// TIA Portal V20 export
DATA_BLOCK "2000_Motion"   // DB450
// stored: MemoryReserve 100
   VAR
      Dancer : Struct
         Commands : Struct
            Enable : Bool;
            Stop : Bool;
            Reset : Bool;
         END_STRUCT;
         Parameters : Struct
            DancerDirection : Bool;
            UnWinderDirection : Bool;
            UnwinderTopUse : Bool;
            UnwinderBottomUse : Bool;
            JogMode : Bool;
            SetPoint : LReal;
            Input : LReal;
            Kp : LReal;
            Ki : LReal;
            Radius : LReal;
         END_STRUCT;
         Status : Struct
            StopRequest : Bool;
            Busy : Struct
               TotalBusy : Bool;
               EnableBusy : Bool;
               StopBusy : Bool;
               ResetBusy : Bool;
            END_STRUCT;
            Done : Struct
               TotalDone : Bool;
               EnableDone : Bool;
               StopDone : Bool;
               ResetDone : Bool;
            END_STRUCT;
            Error : Bool;
            ErrorID : DWord;
            StatusID : DWord;
            NowCmd : DInt;
            BeforeCmd : DInt;
            NowStep : DInt;
            BeforeStep : DInt;
         END_STRUCT;
      END_STRUCT;
      StackMain : Struct
         Commands : Struct
            Calculate : Bool := FALSE;
            SemiStep : Bool := FALSE;
            FullStep : Bool := FALSE;
            Auto : Bool := FALSE;
            CycleStop : Bool := FALSE;
            FastStop : Bool := FALSE;
            Reset : Bool := FALSE;
         END_STRUCT;
         Parameters : Struct
            Global : Struct
               CPM : LReal := 10.0;
               StageWidth : LReal := 244.14;
            END_STRUCT;
            "Step" : Struct
               MandrelUse : Bool;
               InitialPosFinalRoller : LReal := 0.0;
               InitialPosCompensator : LReal := 0.0;
            END_STRUCT;
            Auto : Struct
               SepaClean : Bool;
               CellCount : DInt;
               Compensator : Struct
                  InitialPosCompensator : LReal;
               END_STRUCT;
               Anode : Struct
                  PnPX1 : Struct
                     InitialPosAnodePnPX1 : LReal;
                     AnodePnPX1FwdOutputCam : Struct
                        OnPos : LReal := 10.0;
                        OffPos : LReal := 530.0;
                     END_STRUCT;
                     AnodePnPX1BwdOutputCam : Struct
                        OnPos : LReal := 10.0;
                        OffPos : LReal := 530.0;
                     END_STRUCT;
                     AnodeReelCutDataDeleteOffOutputCam : Struct
                        OnPos : LReal := 10.0;
                        OffPos : LReal := 530.0;
                     END_STRUCT;
                  END_STRUCT;
                  PnPX2 : Struct
                     InitialPosAnodePnPX2 : LReal;
                     AnodePnPX2FwdOutputCam : Struct
                        OnPos : LReal := 10.0;
                        OffPos : LReal := 530.0;
                     END_STRUCT;
                     AnodePnPX2BwdOutputCam : Struct
                        OnPos : LReal := 10.0;
                        OffPos : LReal := 530.0;
                     END_STRUCT;
                  END_STRUCT;
                  PnPZ1 : Struct
                     InitialPosAnodePnPZ1 : LReal := 0.0;
                     AnodePnPZ1Down1OutputCam : Struct
                        OnPos : LReal := 1.0;
                        OffPos : LReal := 24.0;
                     END_STRUCT;
                     AnodePnPZ1Up1OutputCam : Struct
                        OnPos : LReal := 1.0;
                        OffPos : LReal := 24.0;
                     END_STRUCT;
                     AnodePnPZ1Down2OutputCam : Struct
                        OnPos : LReal := 1.0;
                        OffPos : LReal := 29.0;
                     END_STRUCT;
                     AnodePnPZ1Up2OutputCam : Struct
                        OnPos : LReal := 1.0;
                        OffPos : LReal := 29.0;
                     END_STRUCT;
                     AnodePnPZ1SuctionOnOutputCam : Struct
                        OnPos : LReal := 23.0;
                        OffPos : LReal := 28.0;
                     END_STRUCT;
                     AnodePnPZ1SuctionOffOutputCam : Struct
                        OnPos : LReal := 23.0;
                        OffPos : LReal := 30.0;
                     END_STRUCT;
                     AnodePnPZ1ReelCutBlowOutputCam : Struct
                        OnPos : LReal := 22.0;
                        OffPos : LReal := 28.0;
                     END_STRUCT;
                     AnodeAlignSuctionOnOutputCam : Struct
                        OnPos : LReal := 22.0;
                        OffPos : LReal := 30.0;
                     END_STRUCT;
                     AnodeReelCutDataDeleteOnOutputCam : Struct
                        OnPos : LReal := 5.0;
                        OffPos : LReal := 20.0;
                     END_STRUCT;
                     AnodeAlignVisionOutputCam : Struct
                        OnPos : LReal := 1.0;
                        OffPos : LReal := 24.0;
                     END_STRUCT;
                  END_STRUCT;
                  PnPZ2 : Struct
                     InitialPosAnodePnPZ2 : LReal := 0.0;
                     AnodePnPZ2Down1OutputCam : Struct
                        OnPos : LReal := 1.0;
                        OffPos : LReal := 24.0;
                     END_STRUCT;
                     AnodePnPZ2Up1OutputCam : Struct
                        OnPos : LReal := 1.0;
                        OffPos : LReal := 24.0;
                     END_STRUCT;
                     AnodePnPZ2Down2OutputCam : Struct
                        OnPos : LReal := 1.0;
                        OffPos : LReal := 29.0;
                     END_STRUCT;
                     AnodePnPZ2Up2OutputCam : Struct
                        OnPos : LReal := 1.0;
                        OffPos : LReal := 29.0;
                     END_STRUCT;
                     AnodePnPZ2SuctionOnOutputCam : Struct
                        OnPos : LReal := 23.0;
                        OffPos : LReal := 30.0;
                     END_STRUCT;
                     AnodePnPZ2SuctionOffOutputCam : Struct
                        OnPos : LReal := 22.0;
                        OffPos : LReal := 28.0;
                     END_STRUCT;
                     AnodeAlignSuctionOffOutputCam : Struct
                        OnPos : LReal := 22.0;
                        OffPos : LReal := 30.0;
                     END_STRUCT;
                  END_STRUCT;
               END_STRUCT;
               Cathode : Struct
                  PnPX1 : Struct
                     InitialPosCathodePnPX1 : LReal;
                     CathodePnPX1FwdOutputCam : Struct
                        OnPos : LReal := 10.0;
                        OffPos : LReal := 530.0;
                     END_STRUCT;
                     CathodePnPX1BwdOutputCam : Struct
                        OnPos : LReal := 10.0;
                        OffPos : LReal := 530.0;
                     END_STRUCT;
                     CathodeReelCutDataDeleteOffOutputCam : Struct
                        OnPos : LReal := 10.0;
                        OffPos : LReal := 530.0;
                     END_STRUCT;
                  END_STRUCT;
                  PnPX2 : Struct
                     InitialPosCathodePnPX2 : LReal;
                     CathodePnPX2FwdOutputCam : Struct
                        OnPos : LReal := 10.0;
                        OffPos : LReal := 530.0;
                     END_STRUCT;
                     CathodePnPX2BwdOutputCam : Struct
                        OnPos : LReal := 10.0;
                        OffPos : LReal := 530.0;
                     END_STRUCT;
                  END_STRUCT;
                  PnPZ1 : Struct
                     InitialPosCathodePnPZ1 : LReal;
                     CathodePnPZ1Down1OutputCam : Struct
                        OnPos : LReal := 1.0;
                        OffPos : LReal := 24.0;
                     END_STRUCT;
                     CathodePnPZ1Up1OutputCam : Struct
                        OnPos : LReal := 1.0;
                        OffPos : LReal := 24.0;
                     END_STRUCT;
                     CathodePnPZ1Down2OutputCam : Struct
                        OnPos : LReal := 1.0;
                        OffPos : LReal := 29.0;
                     END_STRUCT;
                     CathodePnPZ1Up2OutputCam : Struct
                        OnPos : LReal := 1.0;
                        OffPos : LReal := 29.0;
                     END_STRUCT;
                     CathodePnPZ1SuctionOnOutputCam : Struct
                        OnPos : LReal := 23.0;
                        OffPos : LReal := 28.0;
                     END_STRUCT;
                     CathodePnPZ1SuctionOffOutputCam : Struct
                        OnPos : LReal := 23.0;
                        OffPos : LReal := 30.0;
                     END_STRUCT;
                     CathodePnPZ1ReelCutBlowOutputCam : Struct
                        OnPos : LReal := 22.0;
                        OffPos : LReal := 28.0;
                     END_STRUCT;
                     CathodeAlignSuctionOnOutputCam : Struct
                        OnPos : LReal := 22.0;
                        OffPos : LReal := 30.0;
                     END_STRUCT;
                     CathodeReelCutDataDeleteOnOutputCam : Struct
                        OnPos : LReal := 5.0;
                        OffPos : LReal := 20.0;
                     END_STRUCT;
                     CathodeAlignVisionOutputCam : Struct
                        OnPos : LReal := 1.0;
                        OffPos : LReal := 24.0;
                     END_STRUCT;
                  END_STRUCT;
                  PnPZ2 : Struct
                     InitialPosCathodePnPZ2 : LReal;
                     CathodePnPZ2Down1OutputCam : Struct
                        OnPos : LReal := 1.0;
                        OffPos : LReal := 24.0;
                     END_STRUCT;
                     CathodePnPZ2Up1OutputCam : Struct
                        OnPos : LReal := 1.0;
                        OffPos : LReal := 24.0;
                     END_STRUCT;
                     CathodePnPZ2Down2OutputCam : Struct
                        OnPos : LReal := 1.0;
                        OffPos : LReal := 29.0;
                     END_STRUCT;
                     CathodePnPZ2Up2OutputCam : Struct
                        OnPos : LReal := 1.0;
                        OffPos : LReal := 29.0;
                     END_STRUCT;
                     CathodePnPZ2SuctionOnOutputCam : Struct
                        OnPos : LReal := 23.0;
                        OffPos : LReal := 28.0;
                     END_STRUCT;
                     CathodePnPZ2SuctionOffOutputCam : Struct
                        OnPos : LReal := 23.0;
                        OffPos : LReal := 30.0;
                     END_STRUCT;
                     CathodeAlignSuctionOffOutputCam : Struct
                        OnPos : LReal := 22.0;
                        OffPos : LReal := 30.0;
                     END_STRUCT;
                  END_STRUCT;
               END_STRUCT;
               FinalRoller : Struct
                  InitialPosFinalRoller : LReal;
                  FinalRollerFwdOutputCam : Struct
                     OnPos : LReal := 10.0;
                     OffPos : LReal := 330.0;
                  END_STRUCT;
                  FinalRollerBwdOutputCam : Struct
                     OnPos : LReal := 10.0;
                     OffPos : LReal := 330.0;
                  END_STRUCT;
                  FinalRollerStackTableDownOutputCam : Struct
                     OnPos : LReal := 140.0;
                     OffPos : LReal := 200.0;
                  END_STRUCT;
                  FinalRollerStackAnodeVisionOutputCam : Struct
                     OnPos : LReal := 10.0;
                     OffPos : LReal := 40.0;
                  END_STRUCT;
                  FinalRollerStackCathodeVisionOutputCam : Struct
                     OnPos : LReal := 300.0;
                     OffPos : LReal := 330.0;
                  END_STRUCT;
               END_STRUCT;
               Mandrel : Struct
                  InitialPosAnodeMandrelYFront : LReal;
                  InitialPosAnodeMandrelYRear : LReal;
                  InitialPosAnodeMandrelZFront : LReal;
                  InitialPosAnodeMandrelZRear : LReal;
                  InitialPosCathodeMandrelYFront : LReal;
                  InitialPosCathodeMandrelYRear : LReal;
                  InitialPosCathodeMandrelZFront : LReal;
                  InitialPosCathodeMandrelZRear : LReal;
               END_STRUCT;
            END_STRUCT;
            StackCalculate : Struct
               Direction : Bool := TRUE;
               RatioOption : Bool := TRUE;
               TimeOption : Bool;
               PosOption : Bool;
               DoubleOption : Bool;
               StageHeight : LReal := 360.0;
               StageGap : LReal := 5.0;
               AccRatio : DInt := 3;
               Ratio : Struct
                  FinalRollerStart : LReal := 0.0;
                  FinalRollerEnd : LReal := 75.0;
                  PnPXStart : LReal := 0.0;
                  PnPXEnd : LReal := 75.0;
                  PnPZDownStart : LReal := 65.0;
                  PnPZDownEnd : LReal := 75.0;
                  PnPZUpStart : LReal := 90.0;
                  PnPZUpEnd : LReal := 100.0;
                  MandrelBwdStart : LReal := 75.0;
                  MandrelBwdEnd : LReal := 82.5;
                  MandrelFwdStart : LReal := 82.5;
                  MandrelFwdEnd : LReal := 90.0;
                  MandrelUpStart1 : LReal := 55.0;
                  MandrelUpEnd1 : LReal := 62.5;
                  MandrelUpStart2 : LReal := 75.0;
                  MandrelUpEnd2 : LReal := 82.5;
                  MandrelDownStart : LReal := 87.0;
                  MandrelDownEnd : LReal := 90.0;
                  MandrelYTerm : LReal := 0.0;
                  MandrelZTerm : LReal := 0.0;
                  MandrelBwdOffset : LReal := 0.0;
                  MandrelFwdOffset : LReal := 0.0;
               END_STRUCT;
               "Time" : Struct
                  FinalRollerStart : LReal;
                  FinalRollerEnd : LReal;
                  PnPXStart : LReal;
                  PnPXEnd : LReal;
                  PnPZDownStart : LReal;
                  PnPZDownEnd : LReal;
                  PnPZUpStart : LReal;
                  PnPZUpEnd : LReal;
                  MandrelBwdStart : LReal;
                  MandrelBwdEnd : LReal;
                  MandrelFwdStart : LReal;
                  MandrelFwdEnd : LReal;
                  MandrelUpStart1 : LReal;
                  MandrelUpEnd1 : LReal;
                  MandrelUpStart2 : LReal;
                  MandrelUpEnd2 : LReal;
                  MandrelDownStart : LReal;
                  MandrelDownEnd : LReal;
               END_STRUCT;
               Position : Struct
                  FinalRollerBwdPos : LReal;
                  FinalRollerFwdPos : LReal;
               END_STRUCT;
               Distance : Struct
                  Compensator : Struct
                     Null : Bool;
                  END_STRUCT;
                  Anode : Struct
                     PnPX1Distance : LReal := 540.0;
                     PnPX2Distance : LReal := 540.0;
                     PnPZ1Distance1 : LReal := 25.0;
                     PnPZ1Distance2 : LReal := 27.0;
                     PnPZ2Distance1 : LReal := 25.0;
                     PnPZ2Distance2 : LReal := 27.0;
                  END_STRUCT;
                  Cathode : Struct
                     PnPX1Distance : LReal := 540.0;
                     PnPX2Distance : LReal := 540.0;
                     PnPZ1Distance1 : LReal := 25.0;
                     PnPZ1Distance2 : LReal := 27.0;
                     PnPZ2Distance1 : LReal := 25.0;
                     PnPZ2Distance2 : LReal := 27.0;
                  END_STRUCT;
                  FinalRoller : Struct
                     Distance : LReal := 350.0;
                  END_STRUCT;
                  Mandrel : Struct
                     AnodeMandrelYFrontDistance : LReal := 20.0;
                     AnodeMandrelYRearDistance : LReal := 20.0;
                     CathodeMandrelYFrontDistance : LReal := 20.0;
                     CathodeMandrelYRearDistance : LReal := 20.0;
                     AnodeMandrelZFrontDistance : LReal := 10.0;
                     AnodeMandrelZRearDistance : LReal := 10.0;
                     CathodeMandrelZFrontDistance : LReal := 10.0;
                     CathodeMandrelZRearDistance : LReal := 10.0;
                  END_STRUCT;
               END_STRUCT;
            END_STRUCT;
         END_STRUCT;
         Status : Struct
            StopRequest : Bool;
            Busy : Struct
               TotalBusy : Bool;
               CalculateBusy : Bool;
               SemiStepBusy : Bool;
               FullStepBusy : Bool;
               AutoBusy : Bool;
               CycleStopBusy : Bool;
               FastStopBusy : Bool;
               ResetBusy : Bool;
            END_STRUCT;
            Done : Struct
               TotalDone : Bool;
               CalculateDone : Bool;
               SemiStepDone : Bool;
               FullStepDone : Bool;
               AutoDone : Bool;
               CycleStopDone : Bool;
               FastStopDone : Bool;
               ResetDone : Bool;
            END_STRUCT;
            Error : Bool;
            ErrorID : DWord;
            StatusID : DWord;
            NowCmd : DInt;
            BeforeCmd : DInt;
            NowStep : DInt;
            BeforeStep : DInt;
         END_STRUCT;
         OutputBits : Struct
            AnodePnP1Suction : Bool;
            AnodePnP1Blow : Bool;
            AnodePnP1ReelCutBlow : Bool;
            AnodePnP1RotaryWork : Bool;
            AnodePnP1RotaryHome : Bool;
            AnodeReelCutDataDelete : Bool;
            AnodePnP2Suction : Bool;
            AnodePnP2Blow : Bool;
            AnodeAlignSuction : Bool;
            AnodeAlignBlow : Bool;
            AnodeAlignVision : Bool;
            CathodePnP1Suction : Bool;
            CathodePnP1Blow : Bool;
            CathodePnP1ReelCutBlow : Bool;
            CathodePnP1RotaryWork : Bool;
            CathodePnP1RotaryHome : Bool;
            CathodeReelCutDataDelete : Bool;
            CathodePnP2Suction : Bool;
            CathodePnP2Blow : Bool;
            CathodeAlignSuction : Bool;
            CathodeAlignBlow : Bool;
            CathodeAlignVision : Bool;
            StackTableZAnodeDown : Bool;
            StackTableZCathodeDown : Bool;
            StackAnodeVision : Bool;
            StackCathodeVision : Bool;
         END_STRUCT;
         OutputData : Struct
            StackCellCount : DInt;
         END_STRUCT;
         CamInterface : Struct
            Execute : Bool;
            Done : Bool;
            Busy : Bool;
            Error : Bool;
            ErrorID : DWord;
            NowCmd : DInt;
            BeforeCmd : DInt;
         END_STRUCT;
         ReelcutInterface : Struct
            AnodeReelcutStandby : Bool;
            AnodeReelcutStart : Bool;
            AnodeReelcutDone : Bool;
            CathodeReelcutStandby : Bool;
            CathodeReelcutStart : Bool;
            CathodeReelcutDone : Bool;
         END_STRUCT;
      END_STRUCT;
   END_VAR
BEGIN
END_DATA_BLOCK
